// TIA Portal V20 export
TYPE "LKinCtrl_TeachKinematics_typeInternalEvents"
// stored: Access Published
   STRUCT
      approachPoint { ExternalAccessible := 'False'; ExternalVisible := 'False'; ExternalWritable := 'False'} : "LKinCtrl_typeApproachPoint";
      openPopUp { ExternalAccessible := 'False'; ExternalVisible := 'False'; ExternalWritable := 'False'} : Bool;
      closePopUp { ExternalAccessible := 'False'; ExternalVisible := 'False'; ExternalWritable := 'False'} : Bool;
   END_STRUCT;
END_TYPE
